// TwinCAT 3 PLC project Plc2
// ProgramVersion: 3.1.4024.0
// libraries:
//   Tc2_Standard, * (Beckhoff Automation GmbH)
//   Tc2_System, * (Beckhoff Automation GmbH)
//   Tc3_Module, * (Beckhoff Automation GmbH)
//   VisuDialogs, * (System)
//   VisuSymbols,3.5.10.0,System
// project tree:
//   Elements/Curtain/ Curtain.TcPOU, CurtainControl.TcPOU, CurtainWithManualCalibration.TcPOU, CurtainWithManualCalibrationControl.TcPOU, CurtainWithSensor.TcPOU, CurtainWithSensorControl.TcPOU, I_Curtain.TcIO
//   Elements/Dimmer/ AnalogDevice.TcPOU, AnalogDeviceControl.TcPOU, I_AnalogDevice.TcIO
//   Elements/FAN/ FourStateDevice.TcPOU, FourStateDeviceControl.TcPOU, I_FourStateDevice.TcIO
//   Elements/Lamp/ DigitalLamp_Wrapper.TcPOU, I_DigitalDevice.TcIO, OnOffDevice.TcPOU, OnOffDeviceControl.TcPOU
//   / GlobalTextList.TcGTLO, PlcTask.TcTTO, Visualization Manager.TcVMO (not stored)
//   PRGs/ MAIN.TcPOU, PRG_Home.TcPOU, PRG_Testing.TcPOU
//   Utility/ RampDown.TcPOU, RampUp.TcPOU, F_Scaling.TcPOU
//   z_Trash/ AnalogDeviceControl_1.TcPOU, AnalogDevice_1.TcPOU, DigitalLampWithPushButton_1.TcPOU
//   VISUs/ V_Main.TcVIS
// (motion and I/O tree: see PLC project plc)
// real-time tasks:
//   TASK PlcTask: cycle T#10ms, priority 20, ADS port 350
//   TASK PlcTask1: cycle T#10ms, priority 21, ADS port 351

CONFIGURATION Plc2
    RESOURCE PLC ON TwinCAT3
        TASK PlcTask(INTERVAL := T#10ms, PRIORITY := 21);
        PROGRAM MAIN WITH PlcTask : MAIN;
    END_RESOURCE
END_CONFIGURATION

// ---- Elements/Curtain/I_Curtain.TcIO
INTERFACE I_Curtain

METHOD Close : BOOL
VAR_INPUT
	IN: BOOL;
END_VAR
END_METHOD

METHOD Open : BOOL
VAR_INPUT
	IN: BOOL;
END_VAR
END_METHOD

END_INTERFACE

// ---- Elements/Dimmer/I_AnalogDevice.TcIO
INTERFACE I_AnalogDevice

METHOD DecreaseValue
VAR_INPUT
	EN			: BOOL;
	RampDownTime: TIME;
END_VAR
END_METHOD

METHOD IncreaseValue
VAR_INPUT
	EN			: BOOL;
	RampUpTime: TIME;
END_VAR
END_METHOD

METHOD Off
VAR_INPUT
END_VAR
END_METHOD

METHOD On
VAR_INPUT
END_VAR
END_METHOD

METHOD SetValue
VAR_INPUT
	value: INT;

END_VAR
END_METHOD

PROPERTY Status : INT
GET
END_GET
END_PROPERTY

END_INTERFACE

// ---- Elements/FAN/I_FourStateDevice.TcIO
INTERFACE I_FourStateDevice

METHOD Off
VAR_INPUT
END_VAR
END_METHOD

METHOD On
VAR_INPUT
END_VAR
END_METHOD

METHOD State_1
VAR_INPUT
END_VAR
END_METHOD

METHOD State_2
VAR_INPUT
END_VAR
END_METHOD

METHOD State_3
VAR_INPUT
END_VAR
END_METHOD

METHOD State_4
VAR_INPUT
END_VAR
END_METHOD

PROPERTY Status : INT
GET
END_GET
END_PROPERTY

END_INTERFACE

// ---- Elements/Lamp/I_DigitalDevice.TcIO
INTERFACE I_DigitalDevice

PROPERTY Status : BOOL
GET
END_GET
END_PROPERTY

METHOD TurnOff
VAR_INPUT
END_VAR
END_METHOD

METHOD TurnOn
VAR_INPUT
END_VAR
END_METHOD

END_INTERFACE

// ---- PRGs/MAIN.TcPOU
PROGRAM MAIN
VAR
END_VAR


	PRG_Home();
	PRG_Testing();

END_PROGRAM

// ---- PRGs/PRG_Home.TcPOU
PROGRAM PRG_Home
VAR
	Lamp01	: OnOffDeviceControl;
	Lamp02	: OnOffDeviceControl;
	
	dimmer	: AnalogDeviceControl(ZeroIn:= 0, ZeroOut:= 100, SpanIn:= 0, SpanOut:= 32767, PLC_CYCLE_TIME_ms:= 10, T_LONG_PRESS:= T#2S, RampUpTime:= T#5S, RampDownTime:= T#5S);
	
	fan 	: FourStateDeviceControl;
	
	curtain_basic: CurtainControl;
	curtainWithSensor: CurtainWithSensorControl;
	CurtainWithManualCalibration: CurtainWithManualCalibrationControl(TRUE);
END_VAR


	Lamp01();
	Lamp02();
	
	dimmer();

	fan();

	curtain_basic();
	curtainWithSensor();
	CurtainWithManualCalibration();

END_PROGRAM

// ---- Elements/Lamp/OnOffDeviceControl.TcPOU
FUNCTION_BLOCK OnOffDeviceControl
VAR
	IN AT%I* : BOOL;
	App_OnOff: BOOL;
	digitalLamp : OnOffDevice;	
	rtIN: R_TRIG;
	rtApp_IN: R_TRIG;
END_VAR

	rtIN(CLK:= IN, Q=> );
	rtApp_IN(CLK:= App_OnOff, Q=> );
	
	IF rtIN.Q THEN
		IF digitalLamp.Status = TRUE THEN
			digitalLamp.TurnOff();
		ELSE
			digitalLamp.TurnOn();
		END_IF
	END_IF

	IF rtApp_IN.Q THEN
		IF digitalLamp.Status = TRUE THEN
			digitalLamp.TurnOff();
		ELSE
			digitalLamp.TurnOn();
		END_IF
	END_IF

PROPERTY Status : BOOL
GET
Status	:=	digitalLamp.Status;
END_GET
END_PROPERTY

END_FUNCTION_BLOCK

// ---- Elements/Lamp/OnOffDevice.TcPOU
FUNCTION_BLOCK OnOffDevice IMPLEMENTS I_DigitalDevice
VAR
	Q AT%Q* : BOOL;
END_VAR

PROPERTY Status : BOOL
GET

	Status	:=	Q;
END_GET
END_PROPERTY

METHOD TurnOff
VAR_INPUT
END_VAR

	Q	:=	FALSE;
END_METHOD

METHOD TurnOn
VAR_INPUT
END_VAR

	Q	:=	TRUE;
END_METHOD

END_FUNCTION_BLOCK

// ---- Elements/Dimmer/AnalogDeviceControl.TcPOU
FUNCTION_BLOCK AnalogDeviceControl EXTENDS AnalogDevice
VAR
	On_Inc AT%I* : BOOL;
	Off_Dec AT%I* : BOOL;
	
	App_OnOff: BOOL;
	App_Inc: BOOL;
	App_Dec: BOOL;
	App_SetValue: INT;

	step: INT;
	tonLongPress_01: TON;
	tonLongPress_02: TON;
	_T_LONG_PRESS: TIME;
	_RampUpTime: TIME;
	_RampDownTime: TIME;
	rtOn_Inc: R_TRIG;
	rtOff_Inc: R_TRIG;
	rtApp_Inc: R_TRIG;
	rtApp_Dec: R_TRIG;
	rtApp_OnOff: R_TRIG;
	App_SetValue_prev: INT;
END_VAR


	SUPER^();
	
	rtOn_Inc(CLK:= On_Inc, Q=> );
	rtOff_Inc(CLK:= Off_Dec, Q=> );
	rtApp_OnOff(CLK:= App_OnOff, Q=> );
	rtApp_Inc(CLK:= App_Inc, Q=> );
	rtApp_Dec(CLK:= App_Dec, Q=> );

	CASE step OF
	0:	//	Key pressed
		IF rtOn_Inc.Q THEN
			step := 10;
		ELSIF rtOff_Inc.Q THEN
			step := 50;
		ELSIF rtApp_OnOff.Q THEN
			step	:=	70;	
		ELSIF rtApp_Inc.Q THEN
			step	:=	80;
		ELSIF rtApp_Dec.Q THEN
			step	:=	90;
		ELSIF (App_SetValue_prev <> App_SetValue) THEN
			step	:=	100;
		END_IF
		tonLongPress_01(IN := FALSE);
		tonLongPress_02(IN := FALSE);
		IncreaseValue(FALSE, _RampUpTime);
		DecreaseValue(FALSE, _RampDownTime);
		App_SetValue_prev	:=	App_SetValue;		
		
	10:	//	Short Press - On
		tonLongPress_01(IN:= On_Inc, PT:= _T_LONG_PRESS, Q=> , ET=> );
		IF tonLongPress_01.Q THEN
			step :=	20;
		ELSIF (NOT On_Inc) THEN
			SetValue(value:= REAL_TO_INT(_zeroOut));
			step		:=	0;
		END_IF
		App_SetValue		:=	App_SetValue_prev;
		
	20: // Long Press - Up
		IncreaseValue(TRUE, _RampUpTime);		
			
		IF (NOT On_Inc) THEN
			step	:=	0;
		END_IF
		App_SetValue		:=	App_SetValue_prev;
		
	50:	//	Short press - Off
		tonLongPress_02(IN:= Off_Dec, PT:= _T_LONG_PRESS, Q=> , ET=> );
		IF tonLongPress_02.Q THEN
			step :=	60;
		ELSIF (NOT Off_Dec) THEN
			SetValue(value:= REAL_TO_INT(_zeroIn));
			step		:=	0;
		END_IF
		App_SetValue		:=	App_SetValue_prev;
		
	60:	//	Long press - Down
		DecreaseValue(TRUE, _RampDownTime);
		
		IF (NOT Off_Dec) THEN
			step	:=	0;
		END_IF
		App_SetValue		:=	App_SetValue_prev;
		
	70:
		IF Status <> _zeroIn THEN
			Off();
		ELSE
			On();	
		END_IF
		step	:=	0;
		App_SetValue		:=	App_SetValue_prev;
		
	80:
		IncreaseValue(TRUE, _RampUpTime);		
			
		IF (NOT App_Inc) THEN
			step	:=	0;
		END_IF
		App_SetValue		:=	App_SetValue_prev;
		
	90:
		DecreaseValue(TRUE, _RampDownTime);
		
		IF (NOT App_Dec) THEN
			step	:=	0;
		END_IF
		App_SetValue		:=	App_SetValue_prev;
		
	100:
		SetValue(value:= App_SetValue);
		App_SetValue		:=	App_SetValue_prev;
		step				:=	0;
	END_CASE

METHOD FB_init : BOOL
VAR_INPUT
	bInitRetains : BOOL; // if TRUE, the retain variables are initialized (warm start / cold start)
	bInCopyCode : BOOL;  // if TRUE, the instance afterwards gets moved into the copy code (online change)

	ZeroIn		: REAL;
	ZeroOut    : REAL;
	SpanIn     : REAL;
	SpanOut    : REAL;	
	PLC_CYCLE_TIME_ms: REAL;
	
	T_LONG_PRESS: TIME;
	RampUpTime: TIME;
	RampDownTime: TIME;

	
END_VAR

	//SUPER^.FB_Init(bInitRetains, bInCopyCode, ZeroIn, ZeroOut, SpanIn, SpanOut, PLC_CYCLE_TIME_ms);
	
	_T_LONG_PRESS	:=	T_LONG_PRESS;
	_RampUpTime		:=	RampUpTime;
	_RampDownTime	:=	RampDownTime;
END_METHOD

END_FUNCTION_BLOCK

// ---- Elements/Dimmer/AnalogDevice.TcPOU
FUNCTION_BLOCK AnalogDevice IMPLEMENTS I_AnalogDevice
VAR
	Q AT%Q* : INT;
	rampUp		: RampUp;
	rampDown	: RampDown;
	_value		: REAL;
	_zeroIn		: REAL;
	_zeroOut    : REAL;
	_spanIn     : REAL;
	_spanOut    : REAL;
	_PLC_CYCLE_TIME_ms	: REAL;
	
END_VAR


	Q	:=	REAL_TO_INT(_value);

METHOD DecreaseValue
VAR_INPUT
	EN			: BOOL;
	RampDownTime: TIME;
END_VAR

	rampDown(
		IN					:= EN, 
		RampDownTime		:= RampDownTime, 
		Ramp_lowerLimit		:= _spanIn, 
		Ramp_upperLimit		:= _spanOut, 
		PLC_CYCLE_TIME_ms	:= _PLC_CYCLE_TIME_ms,
		output				:= _value, 
		InProgress			=> );
END_METHOD

METHOD FB_init : BOOL
VAR_INPUT
	bInitRetains : BOOL; // if TRUE, the retain variables are initialized (warm start / cold start)
	bInCopyCode : BOOL;  // if TRUE, the instance afterwards gets moved into the copy code (online change)
	ZeroIn		: REAL;
	ZeroOut    : REAL;
	SpanIn     : REAL;
	SpanOut    : REAL;	
	PLC_CYCLE_TIME_ms: REAL;
END_VAR

	_zeroIn		:=	ZeroIn;
	_zeroOut    :=	ZeroOut;
	_spanIn     :=	SpanIn;
	_spanOut    :=	SpanOut;
	_PLC_CYCLE_TIME_ms	:=	PLC_CYCLE_TIME_ms;
END_METHOD

METHOD IncreaseValue
VAR_INPUT
	EN			: BOOL;
	RampUpTime	: TIME;
END_VAR

	rampUp(
		IN					:= EN, 
		RampUpTime			:= RampUpTime, 
		Ramp_lowerLimit		:= _spanIn, 
		Ramp_upperLimit		:= _spanOut, 
		PLC_CYCLE_TIME_ms	:= _PLC_CYCLE_TIME_ms,
		output				:= _value, 
		InProgress			=> );
END_METHOD

METHOD Off
VAR_INPUT
END_VAR

	_value	:=	_spanIn;
END_METHOD

METHOD On
VAR_INPUT
END_VAR

	_value	:=	_spanOut;
END_METHOD

METHOD SetValue
VAR_INPUT
	value: INT;

END_VAR
	_value	:=	F_Scaling(Variable_In:= value, Input_min:= _zeroIn, Input_max:= _zeroOut, Output_min:= _spanIn, Output_max:= _spanOut);
END_METHOD

PROPERTY Status : INT
GET

	Status	:=	REAL_TO_INT(F_Scaling(Variable_In:= _value, Input_min:= _spanIn, Input_max:= _spanOut, Output_min:= _zeroIn, Output_max:= _zeroOut));
END_GET
END_PROPERTY

END_FUNCTION_BLOCK

// ---- Utility/RampUp.TcPOU
FUNCTION_BLOCK RampUp
VAR_INPUT
	IN: BOOL;
	RampUpTime: TIME;
	Ramp_lowerLimit: REAL;
	Ramp_upperLimit: REAL;
	PLC_CYCLE_TIME_ms: REAL;
END_VAR
VAR_IN_OUT
	output: REAL;
END_VAR
VAR_OUTPUT
	InProgress: BOOL;	
END_VAR
VAR
	rampUp: REAL;
	x: REAL;
	init: BOOL;
END_VAR


	IF IN AND (RampUpTime > T#0S) AND (PLC_CYCLE_TIME_ms > 0) THEN
		IF NOT init THEN
			init	:=	TRUE;
			InProgress	:=	TRUE;
			rampUp	:=	TIME_TO_REAL(RampUpTime);		
			x		:=	PLC_CYCLE_TIME_ms / rampUp;
			x		:=	(Ramp_upperLimit - Ramp_lowerLimit) * x;	
		END_IF
		
		IF (output < Ramp_upperLimit) AND (InProgress) THEN
			output		:=	output + x;
		ELSE
			output		:=	Ramp_upperLimit;
			InProgress	:=	FALSE;
		END_IF
		
	ELSE
		InProgress 	:=	FALSE;	
		init		:=	FALSE;
	END_IF

END_FUNCTION_BLOCK

// ---- Utility/RampDown.TcPOU
FUNCTION_BLOCK RampDown
VAR_INPUT
	IN: BOOL;
	RampDownTime: TIME;
	Ramp_lowerLimit: REAL;
	Ramp_upperLimit: REAL;
	PLC_CYCLE_TIME_ms: REAL;
END_VAR
VAR_IN_OUT
	output: REAL;
END_VAR
VAR_OUTPUT
	InProgress: BOOL;	
END_VAR
VAR
	rampDown: REAL;
	x: REAL;
	init: BOOL;
END_VAR


	IF IN AND (RampDownTime > T#0S) AND (PLC_CYCLE_TIME_ms > 0) THEN
		IF NOT init THEN
			init	:=	TRUE;
			InProgress	:=	TRUE;
			rampDown	:=	TIME_TO_REAL(RampDownTime);		
			x		:=	PLC_CYCLE_TIME_ms / rampDown;
			x		:=	(Ramp_upperLimit - Ramp_lowerLimit) * x;
		END_IF
		
		IF (output > Ramp_lowerLimit) AND (InProgress) THEN
			output		:=	output - x;
		ELSE
			output		:=	Ramp_lowerLimit;
			InProgress	:=	FALSE;
		END_IF
		
	ELSE
		InProgress 	:=	FALSE;	
		init		:=	FALSE;
	END_IF

END_FUNCTION_BLOCK

// ---- Utility/F_Scaling.TcPOU
FUNCTION F_Scaling : REAL
VAR_INPUT
	Variable_In: REAL;			//	raw value of analog card
	Input_min: REAL;			//	min limit of analog card	
	Input_max: REAL;			//	max limit of analog card
	Output_min: REAL;			//	Scalled min limit
	Output_max: REAL;			//	Scalled max limit
END_VAR
VAR
END_VAR


IF (Input_max - Input_min) <> 0 THEN
	F_Scaling := ((Variable_In - Input_min) / (Input_max - Input_min)) * (Output_max - Output_min) + Output_min;
ELSE
	F_Scaling	:=	0;
END_IF


(*
The formula is:
Out := ((Variable_In - ZeroIn) / (SpanIn - ZeroIn)) * (SpanOut - ZeroOut) + ZeroOut.

from chatGPT:
Scaled Value=[(Input Value−Input Min) / (Input Max−Input Min)]×(Output Max−Output Min)+Output Min

Scaling:
(0..100) y = (900..1000)
(a..b) = (y..z)

Ans = (((z-y)/b) * variable) + y
x = (((1000 - 900)/100 ) * y) + 900
*)

END_FUNCTION

// ---- Elements/FAN/FourStateDeviceControl.TcPOU
FUNCTION_BLOCK FourStateDeviceControl EXTENDS FourStateDevice
VAR
	OnOffCmd AT%I* : BOOL;
	
	App_OnOff: BOOL;
	App_FanSpeed: INT;
	
	rtOnOffCmd: R_TRIG;
	rtApp_OnOff: R_TRIG;
	FanSpeed_prev: INT;
END_VAR


	rtOnOffCmd(CLK:= OnOffCmd, Q=> );
	rtApp_OnOff(CLK:= App_OnOff, Q=> );

	IF rtOnOffCmd.Q OR rtApp_OnOff.Q THEN
		IF Status <> 0 THEN
			Off();
		ELSE		
			On();	
		END_IF
	END_IF

	CASE App_FanSpeed OF
		
		0: 	FanSpeed_prev	:=	App_FanSpeed;
		
		1: 	
			IF (FanSpeed_prev <> App_FanSpeed) THEN
				FanSpeed_prev	:=	App_FanSpeed;
				State_1();
			END_IF			
			
		2: 	
			IF (FanSpeed_prev <> App_FanSpeed) THEN
				FanSpeed_prev	:=	App_FanSpeed;
				State_2();
			END_IF			
			
		3: 	
			IF (FanSpeed_prev <> App_FanSpeed) THEN
				FanSpeed_prev	:=	App_FanSpeed;
				State_3();
			END_IF			
			
		4: 	
			IF (FanSpeed_prev <> App_FanSpeed) THEN
				FanSpeed_prev	:=	App_FanSpeed;
				State_4();
			END_IF			
			
	END_CASE

END_FUNCTION_BLOCK

// ---- Elements/FAN/FourStateDevice.TcPOU
FUNCTION_BLOCK FourStateDevice IMPLEMENTS I_FourStateDevice
VAR
	Q	AT%Q* : INT;
	_Status_prev	: INT;
END_VAR

METHOD Off

	Q	:=	REAL_TO_INT(F_Scaling(Variable_In:= 0, Input_min:= 0, Input_max:= 100, Output_min:= 0, Output_max:= 32767));
END_METHOD

METHOD On

	Q	:=	REAL_TO_INT(F_Scaling(Variable_In:= MAX(25, _Status_prev), Input_min:= 0, Input_max:= 100, Output_min:= 0, Output_max:= 32767));
END_METHOD

METHOD State_1

	Q	:=	REAL_TO_INT(F_Scaling(Variable_In:= 25, Input_min:= 0, Input_max:= 100, Output_min:= 0, Output_max:= 32767));
	_Status_prev	:=	25;
END_METHOD

METHOD State_2

	Q	:=	REAL_TO_INT(F_Scaling(Variable_In:= 50, Input_min:= 0, Input_max:= 100, Output_min:= 0, Output_max:= 32767));
	_Status_prev	:=	50;
END_METHOD

METHOD State_3

	Q	:=	REAL_TO_INT(F_Scaling(Variable_In:= 75, Input_min:= 0, Input_max:= 100, Output_min:= 0, Output_max:= 32767));
	_Status_prev	:=	75;
END_METHOD

METHOD State_4

	Q	:=	REAL_TO_INT(F_Scaling(Variable_In:= 100, Input_min:= 0, Input_max:= 100, Output_min:= 0, Output_max:= 32767));
	_Status_prev	:=	100;
END_METHOD

PROPERTY Status : INT
GET

	Status	:=	REAL_TO_INT(F_Scaling(Variable_In:= Q, Input_min:= 0, Input_max:= 32767, Output_min:= 0, Output_max:= 100));
END_GET
END_PROPERTY

END_FUNCTION_BLOCK

// ---- Elements/Curtain/CurtainControl.TcPOU
FUNCTION_BLOCK CurtainControl EXTENDS Curtain
VAR
	OpenCmd AT%I* : BOOL;
	CloseCmd AT%I* : BOOL;
	
	App_OpenCmd: BOOL;
	App_CloseCmd: BOOL;

END_VAR


	IF (OpenCmd OR App_OpenCmd) AND ((NOT CloseCmd) OR (NOT App_CloseCmd)) THEN
		Open(IN	:=	TRUE);
	ELSE
		Open(IN	:=	FALSE);
	END_IF

	IF (CloseCmd OR App_CloseCmd) AND ((NOT OpenCmd) OR (NOT App_OpenCmd)) THEN
		Close(IN	:=	TRUE);
	ELSE
		Close(IN	:=	FALSE);
	END_IF

	IF (OpenCmd AND CloseCmd) OR (App_OpenCmd AND App_CloseCmd) THEN
		Open(IN	:=	FALSE);
		Close(IN	:=	FALSE);
	END_IF

END_FUNCTION_BLOCK

// ---- Elements/Curtain/Curtain.TcPOU
FUNCTION_BLOCK Curtain IMPLEMENTS I_Curtain
VAR
	Open_op AT%Q* : BOOL;
	Close_op AT%Q* : BOOL;

END_VAR

METHOD Close : BOOL
VAR_INPUT
	IN: BOOL;
END_VAR

IF NOT Open_op THEN
	Close_op	:=	IN;
END_IF
END_METHOD

METHOD Open : BOOL
VAR_INPUT
	IN: BOOL;
END_VAR

IF NOT Close_op THEN
	Open_op		:=	IN;
END_IF
END_METHOD

END_FUNCTION_BLOCK

// ---- Elements/Curtain/CurtainWithSensor.TcPOU
FUNCTION_BLOCK CurtainWithSensor EXTENDS Curtain
VAR
	OpenSensor	AT%I* : BOOL;
	CloseSensor	AT%I* : BOOL;

	_OpeningTime: TIME;
	_ClosingTime: TIME;
	_status: REAL;

	M_CalibrationAttempt_open: BOOL;
	M_CalibrationAttempt_close: BOOL;
	tonOpenTimeMeasurement: TON;
	tonCloseTimeMeasurement: TON;
	tonStatusTracker_open: TON;
	tonStatusTracker_close: TON;
	statusTrackerTime: TIME;
	rtIN_open: BOOL;
	rtIN_close: BOOL;
END_VAR

METHOD Close : BOOL
VAR_INPUT
	IN: BOOL;
END_VAR

//	Status - Travel time Calibration (Close Time)
IF OpenSensor AND IN THEN
	M_CalibrationAttempt_close	:=	TRUE;
	tonCloseTimeMeasurement(IN:= FALSE, PT:= T#1D, Q=> , ET=> );
END_IF
IF M_CalibrationAttempt_close AND (NOT OpenSensor) THEN
	toncloseTimeMeasurement(IN:= TRUE, PT:= T#1D, Q=> , ET=> );
END_IF


IF NOT Open_op THEN
	Close_op	:=	IN;

	IF NOT rtIN_close THEN
		rtIN_close			:=	TRUE;		
		statusTrackerTime	:=	REAL_TO_TIME(F_Scaling(Variable_In:= _status, Input_min:= 0, Input_max:= 100, Output_min:= 0, Output_max:= TIME_TO_REAL(_ClosingTime)));			
	END_IF

	tonStatusTracker_close(IN:= close_op, PT:= _closingTime, Q=> , ET=> );
	IF tonStatusTracker_close.IN THEN
		IF statusTrackerTime >= tonStatusTracker_close.ET THEN
			_status	:=	LIMIT( 0, (F_Scaling(Variable_In:= TIME_TO_REAL(statusTrackerTime - tonStatusTracker_close.ET), Input_min:= 0, Input_max:= TIME_TO_REAL(_closingTime), Output_min:= 0, Output_max:= 100)) , 100);
		ELSE
			_status	:=	0;	
		END_IF			
	END_IF
	
END_IF

IF CloseSensor THEN
	Close_op	:=	FALSE;
	
	IF M_CalibrationAttempt_close AND (NOT OpenSensor) THEN
		M_CalibrationAttempt_close	:=	FALSE;
		_ClosingTime			:=	toncloseTimeMeasurement.ET;
		toncloseTimeMeasurement(IN:= FALSE, PT:= T#1D, Q=> , ET=> );
		_status					:=	0;
	END_IF
END_IF

IF (IN = FALSE) THEN
	M_CalibrationAttempt_close	:=	FALSE;
	toncloseTimeMeasurement(IN:= FALSE, PT:= T#1D, Q=> , ET=> );
	tonStatusTracker_close(IN:= FALSE, PT:= , Q=> , ET=> );
	rtIN_close	:=	FALSE;	
END_IF
	
toncloseTimeMeasurement();
tonStatusTracker_close();
END_METHOD

METHOD Open : BOOL
VAR_INPUT
	IN: BOOL;
END_VAR

//	Status - Travel time Calibration (Open Time)
IF CloseSensor AND IN THEN
	M_CalibrationAttempt_open	:=	TRUE;
	tonOpenTimeMeasurement(IN:= FALSE, PT:= T#1D, Q=> , ET=> );
END_IF
IF M_CalibrationAttempt_open AND (NOT CloseSensor) THEN
	tonOpenTimeMeasurement(IN:= TRUE, PT:= T#1D, Q=> , ET=> );
END_IF


IF NOT Close_op THEN
	Open_op	:=	IN;
	
	IF NOT rtIN_open THEN
		rtIN_open			:=	TRUE;
		statusTrackerTime	:=	REAL_TO_TIME(F_Scaling(Variable_In:= _status, Input_min:= 0, Input_max:= 100, Output_min:= 0, Output_max:= TIME_TO_REAL(_OpeningTime)));			
	END_IF

	tonStatusTracker_open(IN:= Open_op, PT:= _OpeningTime, Q=> , ET=> );
	IF tonStatusTracker_open.IN THEN
		IF (tonStatusTracker_open.ET <= _OpeningTime) THEN
			_status	:=	LIMIT( 0, F_Scaling(Variable_In:= TIME_TO_REAL(statusTrackerTime + tonStatusTracker_open.ET), Input_min:= 0, Input_max:= TIME_TO_REAL(_OpeningTime), Output_min:= 0, Output_max:= 100), 100);
		ELSE
			_status	:=	100;	
		END_IF			
	END_IF
		
END_IF

IF OpenSensor THEN
	Open_op	:=	FALSE;
	
	IF M_CalibrationAttempt_open AND (NOT CloseSensor) THEN
		M_CalibrationAttempt_open	:=	FALSE;
		_OpeningTime			:=	tonOpenTimeMeasurement.ET;
		tonOpenTimeMeasurement(IN:= FALSE, PT:= T#1D, Q=> , ET=> );
		_status					:=	100;
	END_IF
END_IF

IF (IN = FALSE) THEN
	M_CalibrationAttempt_open	:=	FALSE;
	tonOpenTimeMeasurement(IN:= FALSE, PT:= T#1D, Q=> , ET=> );
	tonStatusTracker_open(IN:= FALSE, PT:= , Q=> , ET=> );
	rtIN_open	:=	FALSE;
END_IF
	
tonOpenTimeMeasurement();
tonStatusTracker_open();
END_METHOD

PROPERTY Status : INT
GET
Status	:=	REAL_TO_INT(_status);
END_GET
END_PROPERTY

END_FUNCTION_BLOCK

// ---- Elements/Curtain/CurtainWithSensorControl.TcPOU
FUNCTION_BLOCK CurtainWithSensorControl EXTENDS CurtainWithSensor
VAR
	OpenPushButton AT%I* : BOOL;
	ClosePushButton AT%I* : BOOL;
		
	App_OpenPushButton: BOOL;
	App_ClosePushButton: BOOL;
	
	rtOpenPB: R_TRIG;
	rtClosePB: R_TRIG;
	M_OpenCmd: BOOL;
	M_CloseCmd: BOOL;
END_VAR


	rtOpenPB(CLK:= (OpenPushButton OR App_OpenPushButton) AND ((NOT ClosePushButton) OR (NOT App_ClosePushButton)), Q=> );
	rtClosePB(CLK:= (ClosePushButton OR App_ClosePushButton) AND ((NOT OpenPushButton) OR (App_OpenPushButton)), Q=> );

	IF rtOpenPB.Q THEN
		M_OpenCmd	:=	NOT M_OpenCmd;
		IF M_OpenCmd THEN
			Open(IN := TRUE);
		ELSE
			Open(IN := FALSE);	
		END_IF
	END_IF
	IF OpenSensor THEN
		Open(IN := FALSE);
	END_IF
	
	IF rtClosePB.Q THEN
		M_CloseCmd	:=	NOT M_CloseCmd;
		IF M_CloseCmd THEN
			Close(IN := TRUE);
		ELSE
			Close(IN := FALSE);	
		END_IF			
	END_IF
	IF CloseSensor THEN
		Close(IN := FALSE);
	END_IF

END_FUNCTION_BLOCK

// ---- Elements/Curtain/CurtainWithManualCalibration.TcPOU
FUNCTION_BLOCK CurtainWithManualCalibration EXTENDS Curtain
VAR
	_status: REAL;
	_chooseAutoCalibrationAfterReset: BOOL;
	_CalibrationDone: BOOL;
	_OpeningTime: TIME;
	_ClosingTime: TIME;	
	

	tonCalibrationTime: TON;
	tonPowerOnDelay: TON;
	tonClosingTime: TON;
	rtIN_close: BOOL;
	statusTrackerTime: TIME;
	rtIN_open: BOOL;
	tonOpeningTime: TON;
END_VAR


	tonPowerOnDelay(IN:= TRUE, PT:= T#2S, Q=> , ET=> );
	IF tonPowerOnDelay.Q THEN
		Calibration();	
	END_IF

METHOD PRIVATE Calibration : BOOL
VAR_INPUT
END_VAR

	IF NOT _CalibrationDone THEN
		
		IF _chooseAutoCalibrationAfterReset THEN
			Open_op					:=	TRUE;
		END_IF
		
		tonCalibrationTime(IN:= Open_op, PT:= _openingTime, Q=> , ET=> );
		IF tonCalibrationTime.Q THEN
			_status				:=	100;
			_CalibrationDone	:=	TRUE;
			tonCalibrationTime(IN:= FALSE, PT:= _openingTime, Q=> , ET=> );
			Open_op					:=	FALSE;		
		END_IF
	END_IF

	Calibration	:=	_CalibrationDone;
END_METHOD

METHOD Close : BOOL
VAR_INPUT
	IN: BOOL;
END_VAR

	IF NOT Open_op THEN
		Close_op	:=	IN;
		
		IF _CalibrationDone AND (_ClosingTime > T#0S AND _OpeningTime > T#0S) THEN
			IF _status > 0 THEN
				IF NOT rtIN_close THEN
					rtIN_close			:=	TRUE;		
					statusTrackerTime	:=	REAL_TO_TIME(F_Scaling(Variable_In:= _status, Input_min:= 0, Input_max:= 100, Output_min:= 0, Output_max:= TIME_TO_REAL(_ClosingTime)));			
				END_IF		
				tonClosingTime(IN:= TRUE, PT:= _ClosingTime, Q=> , ET=> );
				IF statusTrackerTime >= tonClosingTime.ET THEN
					_status	:=	LIMIT( 0, (F_Scaling(Variable_In:= TIME_TO_REAL(statusTrackerTime - tonClosingTime.ET), Input_min:= 0, Input_max:= TIME_TO_REAL(_closingTime), Output_min:= 0, Output_max:= 100)) , 100);					
				ELSE
					_status			:=	0;
				END_IF					
			ELSE //_status = 0 THEN
				Close_op	:=	FALSE;
				tonClosingTime(IN:= FALSE);
			END_IF
		END_IF	
	ELSE
		Close_op	:=	FALSE;	
	END_IF
		
	IF NOT IN THEN
		rtIN_close	:=	FALSE;
		tonClosingTime(IN:= FALSE);
	END_IF
END_METHOD

PROPERTY ClosingTime : TIME
SET
_closingTime	:=	ClosingTime;
END_SET
END_PROPERTY

METHOD FB_init : BOOL
VAR_INPUT
	bInitRetains : BOOL; // if TRUE, the retain variables are initialized (warm start / cold start)
	bInCopyCode : BOOL;  // if TRUE, the instance afterwards gets moved into the copy code (online change)
	ChooseAutoCalibrationAfterReset: BOOL;
	
END_VAR

	_chooseAutoCalibrationAfterReset	:=	ChooseAutoCalibrationAfterReset;
END_METHOD

METHOD Open : BOOL
VAR_INPUT
	IN: BOOL;
END_VAR

	IF NOT Close_op THEN
		Open_op	:=	IN;
		
		IF _CalibrationDone AND (_ClosingTime > T#0S AND _OpeningTime > T#0S) THEN
			IF _status < 100 THEN
				IF NOT rtIN_open THEN
					rtIN_open			:=	TRUE;		
					statusTrackerTime	:=	REAL_TO_TIME(F_Scaling(Variable_In:= _status, Input_min:= 0, Input_max:= 100, Output_min:= 0, Output_max:= TIME_TO_REAL(_OpeningTime)));			
				END_IF		
				tonOpeningTime(IN:= TRUE, PT:= _OpeningTime, Q=> , ET=> );
				IF (tonOpeningTime.ET <= _OpeningTime) THEN
					_status	:=	LIMIT( 0, (F_Scaling(Variable_In:= TIME_TO_REAL(statusTrackerTime + tonOpeningTime.ET), Input_min:= 0, Input_max:= TIME_TO_REAL(_closingTime), Output_min:= 0, Output_max:= 100)) , 100);
				ELSE
					_status		:=	100;
				END_IF					
			ELSE //_status = 100 THEN
				Open_op		:=	FALSE;
				tonOpeningTime(IN:= FALSE);
			END_IF
		END_IF	
	ELSE
		Open_op		:=	FALSE;	
	END_IF
		
	IF NOT IN THEN
		rtIN_open	:=	FALSE;
		tonOpeningTime(IN:= FALSE);
	END_IF
END_METHOD

PROPERTY OpeningTime : TIME
SET
	_openingTime	:=	OpeningTime;
END_SET
END_PROPERTY

PROPERTY Status : INT
GET

IF _CalibrationDone THEN
	Status	:=	REAL_TO_INT(_status);
ELSE
	Status	:=	0;
END_IF
END_GET
END_PROPERTY

END_FUNCTION_BLOCK

// ---- Elements/Curtain/CurtainWithManualCalibrationControl.TcPOU
FUNCTION_BLOCK CurtainWithManualCalibrationControl EXTENDS CurtainWithManualCalibration
VAR
	OpenPushButton AT%I* : BOOL;
	ClosePushButton AT%I* : BOOL;

	App_OpenPushButton: BOOL;
	App_ClosePushButton: BOOL;
	
	rtOpenPB: R_TRIG;
	rtClosePB: R_TRIG;	
	M_OpenCmd: BOOL;
	M_CloseCmd: BOOL;
END_VAR


	rtOpenPB(CLK:= (OpenPushButton OR App_OpenPushButton) AND ((NOT ClosePushButton) OR (NOT App_ClosePushButton)), Q=> );
	rtClosePB(CLK:= (ClosePushButton OR App_ClosePushButton) AND ((NOT OpenPushButton) OR (App_OpenPushButton)), Q=> );

	IF rtOpenPB.Q THEN
		M_OpenCmd	:=	NOT M_OpenCmd;
		IF M_OpenCmd THEN
			Open(IN := TRUE);
		ELSE
			Open(IN := FALSE);	
		END_IF
	END_IF
	IF Status = 100 THEN
		Open(IN := FALSE);
	END_IF
	
	IF rtClosePB.Q THEN
		M_CloseCmd	:=	NOT M_CloseCmd;
		IF M_CloseCmd THEN
			Close(IN := TRUE);
		ELSE
			Close(IN := FALSE);	
		END_IF			
	END_IF
	IF Status = 0 THEN
		Close(IN := FALSE);
	END_IF

END_FUNCTION_BLOCK

// ---- PRGs/PRG_Testing.TcPOU
PROGRAM PRG_Testing
VAR
	digitalLamp_Wrapper: DigitalLamp_Wrapper;
	digitalLamp_Wrapper2: DigitalLamp_Wrapper;
	
	digitalLampWithPushButton_1: DigitalLampWithPushButton_1;
	digitalLampWithPushButton: OnOffDeviceControl;
	
	analogDevice: AnalogDevice(0, 100, 0, 32767, 10);
	analogStatus: INT;
	setAnalogValue: INT;
	bSetValue: BOOL;
	bInc: BOOL;
	bDec: BOOL;
	bOn: BOOL;
	bOff: BOOL;
	analogDeviceControl: AnalogDeviceControl(ZeroIn:= 0, ZeroOut:= 100, SpanIn:= 0, SpanOut:= 32767, PLC_CYCLE_TIME_ms:= 10, T_LONG_PRESS:= T#2S, RampUpTime:= T#5S, RampDownTime:= T#5S); 
	fan : FourStateDevice;

	fanState: INT := -1;
	fanSpeed: INT;
	
	Variable_In: REAL;			//	raw value of analog card
	Input_min: REAL;			//	min limit of analog card	
	Input_max: REAL;			//	max limit of analog card
	Output_min: REAL;			//	Scalled min limit
	Output_max: REAL;			//	Scalled max limit	
	scalled: REAL;
	
	curtain: Curtain;
	curtainOpening: INT;
	curtainWithSensor: CurtainWithSensor;
	genericCurtain : I_Curtain := CurtainWithSensor;		//	curtain;
	
	bSelectCurtain: BOOL;
	bSelectCurtain2: BOOL;
	simu_tonOpenSensor: TON;
	simu_tonCloseSensor: TON;
	OpenSensor: BOOL;
	CloseSensor: BOOL;
	
	curtainWithManualCalibration: CurtainWithManualCalibration(FALSE);
	simu_Sensor: TIME := T#5s;
END_VAR


	CurtainWithManualCalibration();
	CurtainWithManualCalibration.ClosingTime		:=	simu_Sensor;
	CurtainWithManualCalibration.OpeningTime	:=	simu_Sensor;
	curtainOpening	:=	CurtainWithManualCalibration.Status;
	IF bOn THEN
		CurtainWithManualCalibration.Open(IN := TRUE);
	ELSE
		CurtainWithManualCalibration.Open(IN := FALSE);
	END_IF
	
	IF bOff THEN
		CurtainWithManualCalibration.Close(IN := TRUE);
	ELSE
		CurtainWithManualCalibration.Close(IN := FALSE);
	END_IF	

	
	//CurtainWithSensor(OpenSensor := OpenSensor, CloseSensor := CloseSensor);
//	IF bSelectCurtain THEN
//		genericCurtain	:=	curtain;
//		bSelectCurtain	:=	FALSE;
//	END_IF
//	IF bSelectCurtain2 THEN
//		genericCurtain	:=	curtainWithSensor;
//		bSelectCurtain2	:=	FALSE;
//	END_IF
	
//	curtainOpening	:=	CurtainWithSensor.Status;
//	IF bOn THEN
////		curtain.Open(IN	:=	TRUE);
////		curtainWithSensor.Open(IN	:=	TRUE);
//		genericCurtain.Open(IN	:=	TRUE);
//		simu_tonOpenSensor(IN:= TRUE, PT:= simu_Sensor, Q=> , ET=> );
//		CloseSensor	:= FALSE;
//		IF simu_tonOpenSensor.Q THEN
//			bOn	:=	FALSE;
//			simu_tonOpenSensor(IN:= FALSE);
//			OpenSensor	:=	TRUE;
//		END_IF
//	ELSE
////		curtain.Open(IN	:=	FALSE);
////		curtainWithSensor.Open(IN	:=	FALSE);
//		genericCurtain.Open(IN	:=	FALSE);
//		simu_tonOpenSensor(IN:= FALSE);
//	END_IF
	
//	IF bOff THEN
////		curtain.Close(IN	:=	TRUE);
////		curtainWithSensor.Close(IN	:=	TRUE);
//		genericCurtain.Close(IN	:=	TRUE);
//		simu_tonCloseSensor(IN:= TRUE, PT:= simu_Sensor, Q=> , ET=> );
//		OpenSensor	:=	FALSE;
//		IF simu_tonCloseSensor.Q THEN
//			bOff	:=	FALSE;
//			simu_tonCloseSensor(IN:= FALSE);
//			CloseSensor	:=	TRUE;
//		END_IF
//	ELSE
////		curtain.Close(IN	:=	FALSE);
////		curtainWithSensor.Close(IN	:=	FALSE);
//		genericCurtain.Close(IN	:=	FALSE);
//		simu_tonCloseSensor(IN:= FALSE);
//	END_IF
	


	
//	digitalLamp_Wrapper.KeyType		:=	0;
//	digitalLamp_Wrapper2.KeyType	:=	1;

//	digitalLamp_Wrapper();
//	digitalLamp_Wrapper2();
	
//	digitalLampWithPushButton_1();

//	digitalLampWithPushButton();
	

//	analogDevice();
//	analogStatus	:=	analogDevice.Status;
//	IF bSetValue THEN
//		analogDevice.SetValue(value	:=	setAnalogValue);
//		bSetValue	:=	FALSE;
//	END_IF
	
//	IF bInc THEN
//		analogDevice.IncreaseValue(EN:= TRUE, RampUpTime	:=	T#5S);
//	ELSE
//		analogDevice.IncreaseValue(EN:= FALSE, RampUpTime	:=	T#5S);
//	END_IF
	
//	IF bDec THEN
//		analogDevice.DecreaseValue(EN:= TRUE, RampDownTime	:=	T#5S);
//	ELSE
//		analogDevice.DecreaseValue(EN:= FALSE, RampDownTime	:=	T#5S);
//	END_IF
	
//	IF bOn THEN
//		analogDevice.On();
//	END_IF
	
//	IF bOff THEN
//		analogDevice.Off();
//	END_IF
	
//	analogDeviceControl();
//	analogStatus	:=	analogDeviceControl.Status;
		
//	fan();
//	fanSpeed	:=	fan.Status;
//	IF bOff THEN
//	fan.Off();
//	bOff:=FALSE;
//	END_IF
		
//	IF bOn THEN
//		fan.On();
//		bOn:=FALSE;
//	END_IF
	
//	CASE fanState OF
//	0:	;
//	1:	fan.State_1();
//	2:	fan.State_2();
//	3:	fan.State_3();
//	4:	fan.State_4();
//	END_CASE
	
		
//IF (Input_max - Input_min) <> 0 THEN
//	scalled := ((Variable_In - Input_min) / (Input_max - Input_min)) * (Output_max - Output_min) + Output_min;
//ELSE
//	scalled	:=	0;
//END_IF

END_PROGRAM

// ---- Elements/Lamp/DigitalLamp_Wrapper.TcPOU
FUNCTION_BLOCK DigitalLamp_Wrapper
VAR
	IN AT%I* : BOOL;
	digitalLamp: OnOffDevice;
	_keyType: INT;		//	0: Tap/push button 1: Toggle/latch Button

	rtIN: R_TRIG;
	_app_TurnOn: BOOL;
	rt_app_TurnOn: R_TRIG;
	_app_TurnOff: BOOL;
	rt_app_TurnOff: R_TRIG;
	_app_TurnOnOff: BOOL;
	rt_app_TurnOnOff: R_TRIG;
END_VAR


	IF _keyType = 0 THEN
		rtIN(CLK:= IN, Q=> );
		rt_app_TurnOnOff(CLK:= _app_TurnOnOff, Q=> );
		
		IF rtIN.Q OR rt_app_TurnOnOff.Q THEN
			IF digitalLamp.Status = TRUE THEN
				digitalLamp.TurnOff();
			ELSE
				digitalLamp.TurnOn();	
			END_IF
		END_IF
		
		rt_app_TurnOn(CLK:= _app_TurnOn, Q=> );
		IF rt_app_TurnOn.Q THEN
			digitalLamp.TurnOn();
		END_IF
		rt_app_TurnOff(CLK:= _app_TurnOff, Q=> );
		IF rt_app_TurnOff.Q THEN
			digitalLamp.TurnOff();
		END_IF
		
	ELSIF _keyType = 1 THEN
		IF IN THEN
			digitalLamp.TurnOn();
		ELSE
			digitalLamp.TurnOff();
		END_IF
	ELSE
		digitalLamp.TurnOff();
	END_IF

PROPERTY App_TurnOff : BOOL
SET

	_app_TurnOff :=	App_TurnOff;
END_SET
END_PROPERTY

PROPERTY App_TurnOn : BOOL
SET

	_app_TurnOn :=	App_TurnOn;
END_SET
END_PROPERTY

PROPERTY App_TurnOnOff : BOOL
SET

	_app_TurnOnOff	:=	App_TurnOnOff;
END_SET
END_PROPERTY

PROPERTY KeyType : INT
SET

	_keyType	:=	KeyType;
END_SET
END_PROPERTY

END_FUNCTION_BLOCK

// ---- z_Trash/DigitalLampWithPushButton_1.TcPOU
FUNCTION_BLOCK DigitalLampWithPushButton_1 EXTENDS OnOffDevice
VAR
	IN AT%I* : BOOL;
	
	rtIN: R_TRIG;
END_VAR


	rtIN(CLK:= IN, Q=> );

	IF rtIN.Q THEN
		IF Status = TRUE THEN
			TurnOff();
		ELSE
			TurnOn();
		END_IF
	END_IF

END_FUNCTION_BLOCK

// ---- z_Trash/AnalogDeviceControl_1.TcPOU
FUNCTION_BLOCK AnalogDeviceControl_1
VAR
	On_Inc AT%I* : BOOL;
	Off_Dec AT%I* : BOOL;
	
	_zeroIn		: REAL;
	_zeroOut    : REAL;
	_spanIn     : REAL;
	_spanOut    : REAL;
	_PLC_CYCLE_TIME_ms	: REAL;
	
	analogDevice: AnalogDevice(_zeroIn, _zeroOut, _spanIn, _spanOut, _PLC_CYCLE_TIME_ms);
	App_OnOff: BOOL;
	App_Inc: BOOL;
	App_Dec: BOOL;
	App_SetValue: INT;
	

	
	step: INT;	
	tonLongPress_01: TON;
	tonLongPress_02: TON;
	step: INT;
	dimmer_perc: REAL;
	rampUp: RampUp;
	rampDown: RampDown;	
	_T_LONG_PRESS: TIME;
END_VAR

	
	CASE step OF
	0:	//	Key pressed
		IF On_Inc THEN
			step := 10;
		ELSIF Off_Dec THEN
			step := 50;	
		END_IF
		rampUp(IN := FALSE, output:= dimmer_perc);
		rampDown(In := FALSE, output:= dimmer_perc);
		tonLongPress_01(IN := FALSE);
		tonLongPress_02(IN := FALSE);

	10:	//	Short Press - On
		tonLongPress_01(IN:= On_Inc, PT:= _T_LONG_PRESS, Q=> , ET=> );
		IF tonLongPress_01.Q THEN
			step :=	20;
		ELSIF (NOT On_Inc) THEN
			dimmer_perc	:=	32767;
			step		:=	0;
		END_IF		
		
	20: // Long Press - Up
	
		analogDevice.IncreaseValue(EN:= , RampUpTime:= );
			
		IF (NOT On_Inc) THEN
			step	:=	0;
		END_IF		
		
	END_CASE

METHOD FB_init : BOOL
VAR_INPUT
	bInitRetains : BOOL; // if TRUE, the retain variables are initialized (warm start / cold start)
	bInCopyCode : BOOL;  // if TRUE, the instance afterwards gets moved into the copy code (online change)
	T_LONG_PRESS: TIME;
	ZeroIn		: REAL;
	ZeroOut    : REAL;
	SpanIn     : REAL;
	SpanOut    : REAL;	
	PLC_CYCLE_TIME_ms: REAL;

END_VAR

	_zeroIn		:=	ZeroIn;
	_zeroOut    :=	ZeroOut;
	_spanIn     :=	SpanIn;
	_spanOut    :=	SpanOut;
	_PLC_CYCLE_TIME_ms	:=	PLC_CYCLE_TIME_ms;

	_T_LONG_PRESS	:=	T_LONG_PRESS;
END_METHOD

PROPERTY Status : INT
GET
Status	:=	analogDevice.Status;
END_GET
END_PROPERTY

END_FUNCTION_BLOCK

// ---- z_Trash/AnalogDevice_1.TcPOU
FUNCTION_BLOCK AnalogDevice_1 IMPLEMENTS I_AnalogDevice
VAR
	Q AT%I* : INT;
	rampUp		: RampUp;
	rampDown	: RampDown;
	_value		: REAL;
	_zeroIn		: REAL;
	_zeroOut    : REAL;
	_spanIn     : REAL;
	_spanOut    : REAL;
	_PLC_CYCLE_TIME_ms	: REAL;
	
END_VAR


	Q	:=	REAL_TO_INT(_value);

METHOD DecreaseValue
VAR_INPUT
	EN			: BOOL;
	RampDownTime: TIME;
END_VAR

	rampDown(
		IN					:= EN, 
		RampDownTime		:= RampDownTime, 
		Ramp_lowerLimit		:= _spanIn, 
		Ramp_upperLimit		:= _spanOut, 
		PLC_CYCLE_TIME_ms	:= _PLC_CYCLE_TIME_ms,
		output				:= _value, 
		InProgress			=> );
END_METHOD

METHOD FB_init : BOOL
VAR_INPUT
	bInitRetains : BOOL; // if TRUE, the retain variables are initialized (warm start / cold start)
	bInCopyCode : BOOL;  // if TRUE, the instance afterwards gets moved into the copy code (online change)
	ZeroIn		: REAL;
	ZeroOut    : REAL;
	SpanIn     : REAL;
	SpanOut    : REAL;	
	PLC_CYCLE_TIME_ms: REAL;
END_VAR

	_zeroIn		:=	ZeroIn;
	_zeroOut    :=	ZeroOut;
	_spanIn     :=	SpanIn;
	_spanOut    :=	SpanOut;
	_PLC_CYCLE_TIME_ms	:=	PLC_CYCLE_TIME_ms;
END_METHOD

METHOD IncreaseValue
VAR_INPUT
	EN			: BOOL;
	RampUpTime: TIME;
END_VAR

	rampUp(
		IN					:= EN, 
		RampUpTime			:= RampUpTime, 
		Ramp_lowerLimit		:= _spanIn, 
		Ramp_upperLimit		:= _spanOut, 
		PLC_CYCLE_TIME_ms	:= _PLC_CYCLE_TIME_ms,
		output				:= _value, 
		InProgress			=> );
END_METHOD

METHOD Off
VAR_INPUT
END_VAR

	_value	:=	_spanIn;
END_METHOD

METHOD On
VAR_INPUT
END_VAR

	_value	:=	_spanOut;
END_METHOD

METHOD SetValue
VAR_INPUT
	value: INT;

END_VAR

	_value	:=	F_Scaling(Variable_In:= value, Input_min:= _zeroIn, Input_max:= _zeroOut, Output_min:= _spanIn, Output_max:= _spanOut);
END_METHOD

PROPERTY Status : INT
GET

	Status	:=	REAL_TO_INT(F_Scaling(Variable_In:= _value, Input_min:= _spanIn, Input_max:= _spanOut, Output_min:= _zeroIn, Output_max:= _zeroOut));
END_GET
END_PROPERTY

END_FUNCTION_BLOCK

// ---- GlobalTextList.TcGTLO
TEXTLIST GlobalTextList
  675 = '%d'
  555 = 'Dec'
  265 = 'Home Automation'
  962 = 'Inc'
  240 = 'On / Off'
  277 = 'Status: %d'
END_TEXTLIST

// ---- VISUs/V_Main.TcVIS
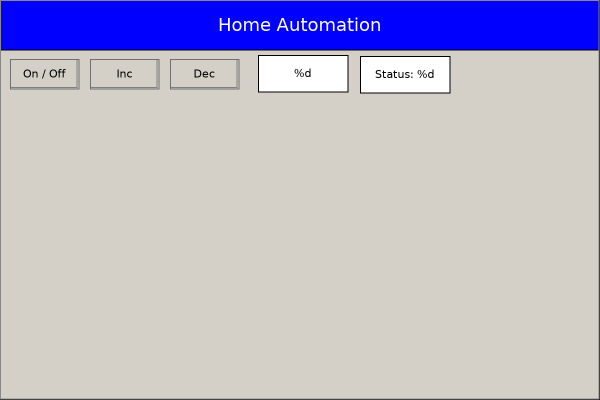
VISUALIZATION V_Main  // 600x400
    Rectangle (0,0 600x400)
    Rectangle (0,0 600x50), "Home Automation"
    Button (10,59 69x30), "On / Off"
        tap PRG_Testing.analogDeviceControl.App_OnOff
    Button (90,59 69x30), "Inc"
        tap PRG_Testing.analogDeviceControl.App_Inc
    Button (170,59 69x30), "Dec"
        tap PRG_Testing.analogDeviceControl.App_Dec
    Rectangle (258,55 90x37), "%d", text variable: PRG_Testing.analogDeviceControl.App_SetValue
        OnMouseClick: write the text variable via VisuDialogs.Numpad, min 0, max 100
    Rectangle (360,56 90x37), "Status: %d", text variable: PRG_Testing.analogStatus
END_VISUALIZATION
